// TIA Portal V15 export
// export: Created 2019-02-11T17:35:22.7858246Z, ExportSetting WithDefaults, WithReadOnly, DisplayName Totally Integrated Automation Portal, DisplayVersion V15 Update 2, DisplayName TIA Portal Openness, DisplayVersion V15 Update 2, DisplayName STEP 7 Professional, DisplayVersion V15 Update 2, DisplayName STEP 7 Safety, DisplayVersion V15, DisplayName WinCC Professional, DisplayVersion V15 Update 2, DisplayName SIMATIC Visualization Architect, DisplayVersion V15 Update 1
DATA_BLOCK "FGDB_ROBNAME@Welding"   // DB36
{ S7_Optimized_Access := 'FALSE' }
AUTHOR : integra
FAMILY : SUB
VERSION : 1.0
// stored: AutoNumber true, CodeModifiedDate 2019-02-11T17:32:00.5944808Z, CompileDate 2019-02-11T17:35:11.3978336Z, CreationDate 2019-02-11T17:32:00.5106573Z, DBAccessibleFromOPCUA true, InstanceOfName iSF_TECH_ROBOT_WELDING, InstanceOfNumber 22, InstanceOfType FB, InterfaceModifiedDate 2018-07-06T04:55:37.0360694Z, IsConsistent true, IsKnowHowProtected false, ModifiedDate 2019-02-11T17:32:00.5944808Z, ParameterModified 2018-07-06T04:51:27.5736649Z, StructureModified 2018-07-06T04:51:27.5736649Z, UDAEnableTagReadback false
"iSF_TECH_ROBOT_WELDING"
   // VAR_INPUT
   //    fct : Int;
   //    safetyStop : Bool;
   //    selectGroupMilling : Bool;
   //    resetAutoTipChange : Bool;
   //    resetManuellTipChange : Bool;
   // END_VAR
   // VAR_OUTPUT
   //    requestGroupMilling : Bool;
   //    requestAutoTipChange : Bool;
   //    requestAutoGroupTipChange : Bool;
   //    requestManuellTipChange : Bool;
   //    requestManuellGroupTipChange : Bool;
   //    reqWaterPumpOn : Bool;
   //    dress1HomePosition : Bool;
   //    dress2HomePosition : Bool;
   //    dress3HomePosition : Bool;
   //    fault : Bool;
   // END_VAR
   // VAR_IN_OUT
   //    IfcFGExternal : "iUDT_IFC_SYS_EXTERNAL_ALARM";
   //    IfcTECH : "iUDT_IFC_ROBOT_TECH";
   //    In_PI_TECH : "iUDT_PI_ROBOT_ADRxx48_TECH";
   //    Out_PO_TECH : "iUDT_PO_ROBOT_ADRxx48_TECH";
   // END_VAR
   // VAR
   //    F : Struct
   //       wrongID : Bool;
   //       notReady : Bool;
   //       powerCircuitBreaker : Bool;
   //       notFI : Bool;
   //       qStop : Bool;
   //       maxTipLifespan : Bool;
   //       motorProtectionTrip : Bool;
   //       fuseFailed : Bool;
   //       coolingWaterError : Bool;
   //       maxLifeCutter : Bool;
   //    END_STRUCT;
   //    Masks : Struct
   //       disableFault1_8 : Byte;
   //       disableFault9_16 : Byte;
   //       prodRelevantFault1_8 : Byte;
   //       prodRelevantFault9_16 : Byte;
   //    END_STRUCT;
   //    LastState : Struct
   //       fault1_8 : Byte;
   //       fault9_16 : Byte;
   //    END_STRUCT;
   //    Tmr : Struct
   //       s1 { S7_SetPoint := 'True'} : Int;
   //       a1 : Int;
   //    END_STRUCT;
   //    VCB : Struct
   //       selectionGroupTipChange : Bool;
   //       selectionGroupMilling : Bool;
   //    END_STRUCT;
   //    TmrB : Struct
   //       "1_EnableDelayTime" : Bool;
   //       "1_RunDelayTime" : Bool;
   //       "1_DoneDelayTime" : Bool;
   //    END_STRUCT;
   //    D : Struct
   //       selectionGroupMilling : Bool;
   //       edgeSelectionGroupMilling : Bool;
   //       autoTipChange : Bool;
   //       autoGroupTipChange : Bool;
   //       manuellTipChange : Bool;
   //       manuellGroupTipChange : Bool;
   //    END_STRUCT;
   //    TECH_IN : Struct
   //       ID : Byte;
   //       ready : Bool;
   //       noEstop : Bool;
   //       userSafeNotDetect : Bool;
   //       drivesOK : Bool;
   //       qStop : Bool;
   //       reqGroupTipChange : Bool;
   //       maxTipLifespan : Bool;
   //       prewarningTipChange : Bool;
   //       reqGroupTipDresser : Bool;
   //       reqTipDresser : Bool;
   //       prewarningTipDresser : Bool;
   //       maxLifeCutter : Bool;
   //       motorProtectionTrip : Bool;
   //       circuitBreakerOn : Bool;
   //       noFaultcurrent : Bool;
   //       fuseFaied : Bool;
   //       dress1WorkPosition : Bool;
   //       dress1HomePosition : Bool;
   //       dress2WorkPosition : Bool;
   //       dress2HomePosition : Bool;
   //       dress3WorkPosition : Bool;
   //       dress3HomePosition : Bool;
   //       tipChangerAvailable : Bool;
   //       magazinWarning : Bool;
   //       magazinEmpty : Bool;
   //       reqWaterPumpOn : Bool;
   //       coolingWaterError : Bool;
   //       technoBit28 : Bool;
   //       technoBit29 : Bool;
   //       technoBit30 : Bool;
   //       technoBit31 : Bool;
   //       technoBit32 : Bool;
   //       technoBit33 : Bool;
   //       technoBit34 : Bool;
   //       technoBit35 : Bool;
   //       technoBit36 : Bool;
   //       technoBit37 : Bool;
   //       technoBit38 : Bool;
   //       technoBit39 : Bool;
   //       technoBit40 : Bool;
   //    END_STRUCT;
   //    TECH_OUT : Struct
   //       ID { ExternalWritable := 'False'} : Byte;
   //       reqGroupTipDress : Bool;
   //       reqGroupTipChange : Bool;
   //       reqAutoCollectivTipChange : Bool;
   //       reqManCollectivTipChange : Bool;
   //       technoBit4 : Bool;
   //       technoBit5 : Bool;
   //       technoBit6 : Bool;
   //       technoBit7 : Bool;
   //       technoBit9 : Bool;
   //       technoBit10 : Bool;
   //       technoBit11 : Bool;
   //       technoBit12 : Bool;
   //       technoBit13 : Bool;
   //       technoBit14 : Bool;
   //       technoBit15 : Bool;
   //       technoBit16 : Bool;
   //       technoBit17 : Bool;
   //       technoBit18 : Bool;
   //       technoBit19 : Bool;
   //       technoBit20 : Bool;
   //       technoBit21 : Bool;
   //       technoBit22 : Bool;
   //       technoBit23 : Bool;
   //       technoBit24 : Bool;
   //       technoBit25 : Bool;
   //       technoBit26 : Bool;
   //       technoBit27 : Bool;
   //       technoBit28 : Bool;
   //       technoBit29 : Bool;
   //       technoBit30 : Bool;
   //       technoBit31 : Bool;
   //       technoBit32 : Bool;
   //       technoBit33 : Bool;
   //       technoBit34 : Bool;
   //       technoBit35 : Bool;
   //       technoBit36 : Bool;
   //       technoBit37 : Bool;
   //       technoBit38 : Bool;
   //       technoBit39 : Bool;
   //       technoBit40 : Bool;
   //    END_STRUCT;
   // END_VAR
BEGIN
END_DATA_BLOCK
